{attribute 'GeneratedUsingTerminal: EL3204-0162-0016'}
{attribute addProperty BoxType "EL3204-0162-0016"}
{attribute addProperty Description "EL3204-0162 2Ch. Ana. In. PT100 (RTD), 2Ch. Ana. In. +/-10V, 0-10V configurable"}
{attribute addProperty Physics "KK"}
{attribute addProperty Id "RTD_Inputs_Channel_1AT %I*AI_Standard_Channel_4A3944819RTD_Inputs_Channel_2AT %I*AI_Standard_Channel_4A3944819AI_Standard_Channel_1AT %I*AI_Standard_Channel_4A3944819AI_Standard_Channel_2AT %I*AI_Standard_Channel_4A3944819WcStateAT %I*WcState_9091E0EB2InfoDataAT %I*InfoData_32EB74EA10"}
{attribute addProperty CRC "2559361572"}
{attribute addProperty Size "48"}
TYPE EL3204_988CC224 EXTENDS EtcSlaveTerminalBase_947E5A46 :
STRUCT
	{attribute addProperty Name "RTD_Inputs_Channel_1"}
	RTD_Inputs_Channel_1 : AI_Standard_Channel_4A394481;
	{attribute addProperty Name "RTD_Inputs_Channel_2"}
	RTD_Inputs_Channel_2 : AI_Standard_Channel_4A394481;
	{attribute addProperty Name "AI_Standard_Channel_1"}
	AI_Standard_Channel_1 : AI_Standard_Channel_4A394481;
	{attribute addProperty Name "AI_Standard_Channel_2"}
	AI_Standard_Channel_2 : AI_Standard_Channel_4A394481;
	{attribute addProperty Name "WcState"}
	WcState : WcState_9091E0EB;
	{attribute addProperty Name "InfoData"}
	InfoData : InfoData_32EB74EA;
END_STRUCT
END_TYPE

(* stored: Version 1.2.0.0, ProductVersion 3.1.4024.11
   DUT EL3204_988CC224: Id {6983a1e7-1b3c-49c5-8541-736b05591183} *)
